KUKA KRL program: Grp_sps.sub

&ACCESS RVO
&COMMENT GripperTech PLC program
DEF  Grp_sps ( )

  LOOP
    Grp_MonPLC()
  ENDLOOP
  ;FOLD ;%{H};
    END
  ;ENDFOLD
